KUKA KRL program: fork_close_test.src, fork_close_test.dat

--- fork_close_test.src ---
&ACCESS RVO
&REL 5
&PARAM DISKPATH = Program/iPower
DEF  fork_close_test ( )
   ;FOLD INI;%{PE}
      ;FOLD BASISTECH INI
         GLOBAL INTERRUPT DECL 3 WHEN $STOPMESS==TRUE DO IR_STOPM ( )
         INTERRUPT ON 3
         BAS (#INITMOV,0 )
      ;ENDFOLD (BASISTECH INI)
      ;FOLD USER INI
         ;Make your modifications here

      ;ENDFOLD (USER INI)
   ;ENDFOLD (INI)
   $PAL_MODE = TRUE

;FOLD PTP P2 Vel=100 % PDAT2 Tool[1] Base[0];%{PE}%R 8.3.44,%MKUKATPBASIS,%CMOVE,%VPTP,%P 1:PTP, 2:P2, 3:, 5:100, 7:PDAT2
$BWDSTART=FALSE
PDAT_ACT=PPDAT2
FDAT_ACT=FP2
BAS(#PTP_PARAMS,100)
PTP XP2
;ENDFOLD
   LOOP
      ARTForkClose(1)
      ;doGripCloseFork = FALSE
      WAIT SEC 10
      ARTForkClose(2)
      ;doGripCloseFork = FALSE
      WAIT SEC 10
      ARTForkOpen()
      WAIT SEC 10
   ENDLOOP

END

--- fork_close_test.dat ---
&ACCESS RVO
&REL 5
&PARAM DISKPATH = Program/iPower
DEFDAT  fork_close_test
;FOLD EXTERNAL DECLARATIONS;%{PE}%MKUKATPBASIS,%CEXT,%VCOMMON,%P
;FOLD BASISTECH EXT;%{PE}%MKUKATPBASIS,%CEXT,%VEXT,%P
EXT  BAS (BAS_COMMAND  :IN,REAL  :IN )
;ENDFOLD (BASISTECH EXT)
;FOLD USER EXT;%{E}%MKUKATPUSER,%CEXT,%VEXT,%P
;Make your modifications here

;ENDFOLD (USER EXT)
;ENDFOLD (EXTERNAL DECLARATIONS)
DECL BASIS_SUGG_T LAST_BASIS={POINT1[] "P2                      ",POINT2[] "P2                      ",CP_PARAMS[] "CPDAT0                  ",PTP_PARAMS[] "PDAT2                   ",CONT[] "                        ",CP_VEL[] "2.0                     ",PTP_VEL[] "100                     ",SYNC_PARAMS[] "SYNCDAT                 ",SPL_NAME[] "S0                      ",A_PARAMS[] "ADAT0                   "}
DECL E6POS XP1={X -1475.37585,Y -275.516022,Z 1472.78064,A -64.4847794,B 87.3439941,C 27.0488091,S 6,T 50,E1 0.0,E2 0.0,E3 0.0,E4 0.0,E5 0.0,E6 0.0}
DECL FDAT FP1={TOOL_NO 1,BASE_NO 0,IPO_FRAME #BASE,POINT2[] " ",TQ_STATE FALSE}
DECL PDAT PPDAT1={VEL 100.000,ACC 100.000,APO_DIST 100.000,GEAR_JERK 50.0000,EXAX_IGN 0}
DECL E6POS XP2={X 934.834534,Y -775.734802,Z 1807.41467,A 96.2909927,B 1.31615803E-08,C 180.000,S 2,T 42,E1 0.0,E2 0.0,E3 0.0,E4 0.0,E5 0.0,E6 0.0}
DECL FDAT FP2={TOOL_NO 1,BASE_NO 0,IPO_FRAME #BASE,POINT2[] " ",TQ_STATE FALSE}
DECL PDAT PPDAT2={VEL 100.000,ACC 100.000,APO_DIST 100.000,GEAR_JERK 50.0000,EXAX_IGN 0}
ENDDAT
